(* PLC project Beremiz Python Support Tests, LOLITECH Beremiz 0.0 *)
(* stored: creationDateTime 2008-12-14 16:21:19, modificationDateTime 2009-01-19 09:02:00 *)

PROGRAM main_pytest
  VAR
    pytest_var1 : STRING;
    pytest_var2 : BOOL;
    py2 : python_poll;
    py3 : python_poll;
    py1 : python_poll;
    pytest_var3 : BOOL;
    pollX : python_poll;
    pollY : python_poll;
  END_VAR
  VAR  (* added by the conversion: wires and edge detectors of the diagram *)
    _STRING_TO_UINT24_ENO : BOOL;
    _STRING_TO_UINT24_OUT : UINT;
    _UINT_TO_BOOL25_OUT : BOOL;
    _STRING_TO_INT43_ENO : BOOL;
    _STRING_TO_INT43_OUT : INT;
    _INT_TO_STRING44_ENO : BOOL;
    _INT_TO_STRING44_OUT : STRING;
    _CONCAT42_ENO : BOOL;
    _CONCAT42_OUT : STRING;
    _STRING_TO_INT50_ENO : BOOL;
    _STRING_TO_INT50_OUT : INT;
    _INT_TO_STRING49_ENO : BOOL;
    _INT_TO_STRING49_OUT : STRING;
    _CONCAT48_ENO : BOOL;
    _CONCAT48_OUT : STRING;
  END_VAR

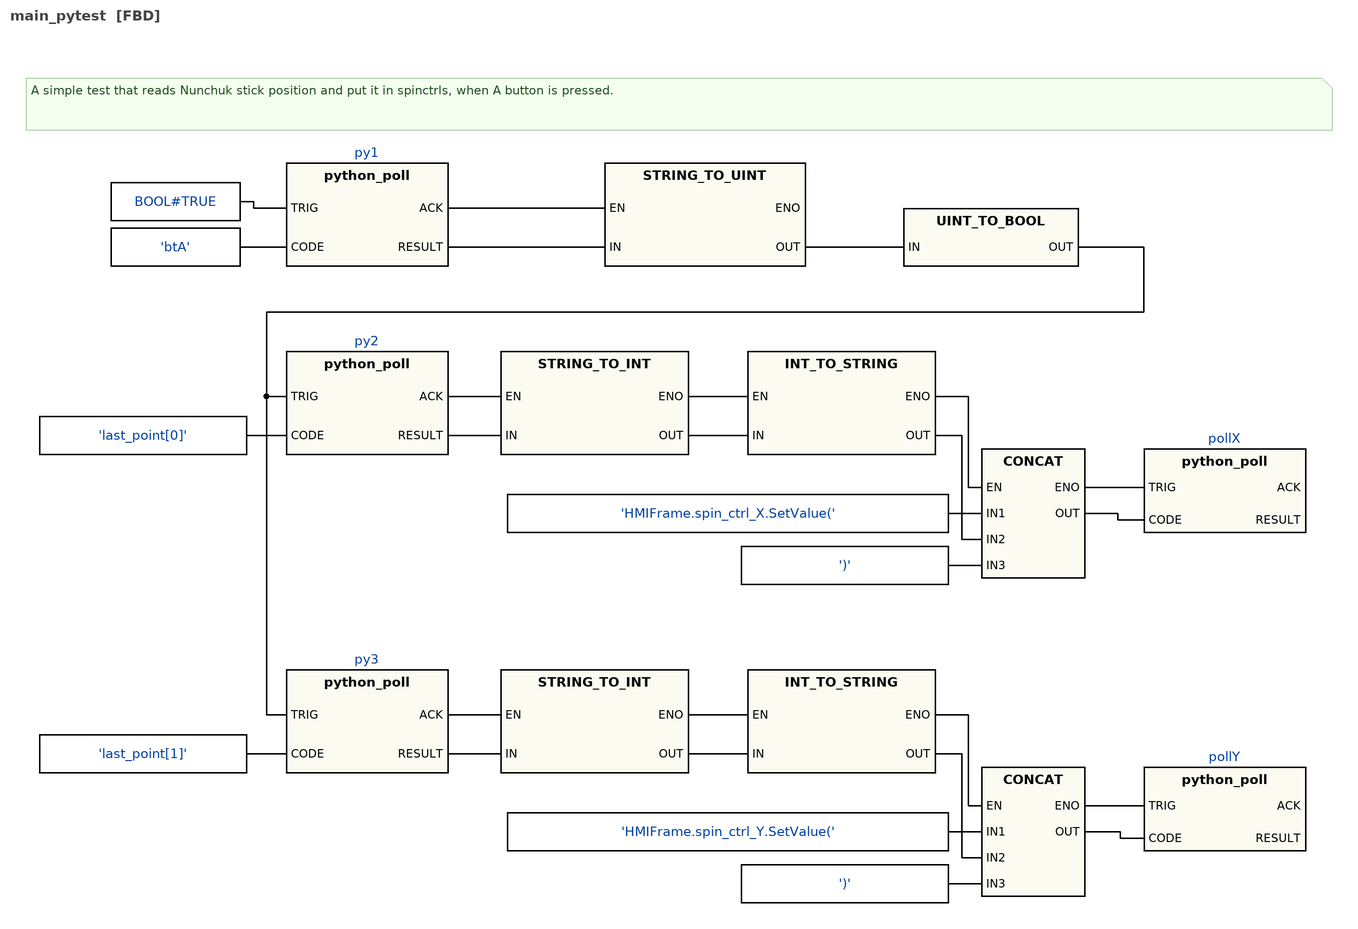
(* FBD diagram, written out as Structured Text *)
(* A simple test that reads Nunchuk stick position and put it in spinctrls, when A button is pressed. *)
py1(TRIG := BOOL#TRUE, CODE := 'btA');
_STRING_TO_UINT24_OUT := STRING_TO_UINT(EN := py1.ACK, IN := py1.RESULT, ENO => _STRING_TO_UINT24_ENO);
_UINT_TO_BOOL25_OUT := UINT_TO_BOOL(_STRING_TO_UINT24_OUT);
py2(TRIG := _UINT_TO_BOOL25_OUT, CODE := 'last_point[0]');
_STRING_TO_INT43_OUT := STRING_TO_INT(EN := py2.ACK, IN := py2.RESULT, ENO => _STRING_TO_INT43_ENO);
_INT_TO_STRING44_OUT := INT_TO_STRING(EN := _STRING_TO_INT43_ENO, IN := _STRING_TO_INT43_OUT, ENO => _INT_TO_STRING44_ENO);
_CONCAT42_OUT := CONCAT(EN := _INT_TO_STRING44_ENO, IN1 := 'HMIFrame.spin_ctrl_X.SetValue(', IN2 := _INT_TO_STRING44_OUT, IN3 := ')', ENO => _CONCAT42_ENO);
pollX(TRIG := _CONCAT42_ENO, CODE := _CONCAT42_OUT);
py3(TRIG := _UINT_TO_BOOL25_OUT, CODE := 'last_point[1]');
_STRING_TO_INT50_OUT := STRING_TO_INT(EN := py3.ACK, IN := py3.RESULT, ENO => _STRING_TO_INT50_ENO);
_INT_TO_STRING49_OUT := INT_TO_STRING(EN := _STRING_TO_INT50_ENO, IN := _STRING_TO_INT50_OUT, ENO => _INT_TO_STRING49_ENO);
_CONCAT48_OUT := CONCAT(EN := _INT_TO_STRING49_ENO, IN1 := 'HMIFrame.spin_ctrl_Y.SetValue(', IN2 := _INT_TO_STRING49_OUT, IN3 := ')', ENO => _CONCAT48_ENO);
pollY(TRIG := _CONCAT48_ENO, CODE := _CONCAT48_OUT);
END_PROGRAM

CONFIGURATION conf_pytest
  RESOURCE res_pytest ON PLC
    TASK pytest_task(INTERVAL := 00:00:00.100000, PRIORITY := 0);
    PROGRAM pytest_instance : main_pytest;
  END_RESOURCE
END_CONFIGURATION
